SUBAPPLICATION SRV_CLIENT (* ROS 2 SRV Client *)
  (* Standard: 61499-2 *)
  (* Version 1.0, 2023-03-14, Tim Hesse *)
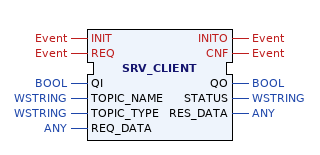
  EVENT_INPUT
    INIT; (* Initialization Request *)
    REQ; (* Normal Execution Request *)
  END_EVENT
  EVENT_OUTPUT
    INITO; (* Initialization Confirm *)
    CNF; (* Execution Confirmation *)
  END_EVENT
  VAR_INPUT
    QI : BOOL; (* Input event qualifier *)
    TOPIC_NAME : WSTRING; (* ROS 2 Topic Name *)
    TOPIC_TYPE : WSTRING; (* ROS 2 Topic Type *)
    REQ_DATA : ANY; (* Request Data *)
  END_VAR
  VAR_OUTPUT
    QO : BOOL; (* Output Event Qualifier *)
    STATUS : WSTRING; (* Service Status *)
    RES_DATA : ANY; (* Response Data *)
  END_VAR
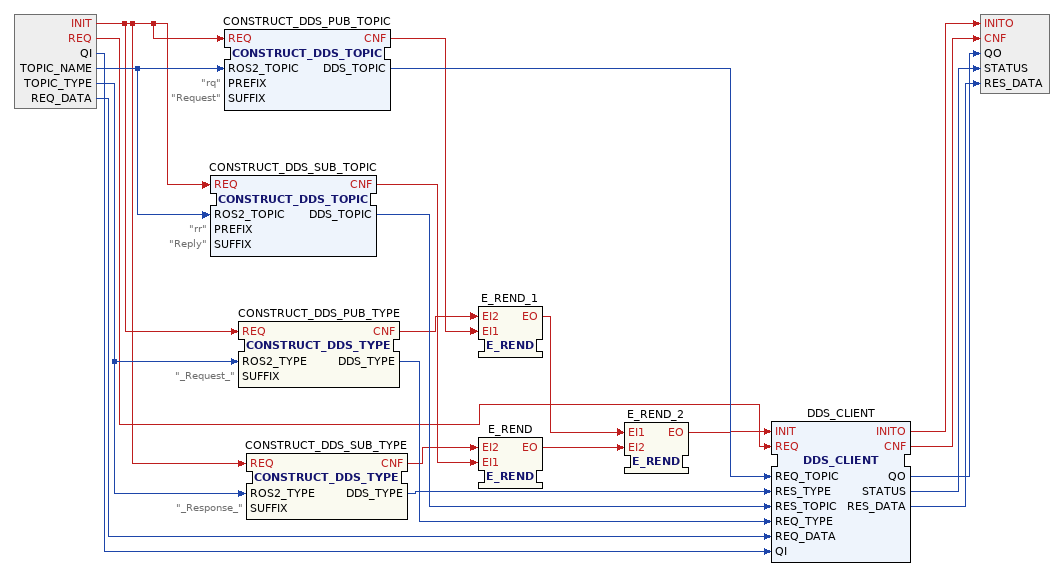
  FBS
    CONSTRUCT_DDS_PUB_TYPE : CONSTRUCT_DDS_TYPE(SUFFIX := "_Request_");
    CONSTRUCT_DDS_SUB_TYPE : CONSTRUCT_DDS_TYPE(SUFFIX := "_Response_");
    E_REND : E_REND;
    E_REND_1 : E_REND;
    E_REND_2 : E_REND;
  END_FBS
  SUBAPPS
    CONSTRUCT_DDS_PUB_TOPIC : CONSTRUCT_DDS_TOPIC(PREFIX := "rq", SUFFIX := "Request");
    CONSTRUCT_DDS_SUB_TOPIC : CONSTRUCT_DDS_TOPIC(PREFIX := "rr", SUFFIX := "Reply");
    DDS_CLIENT : DDS_CLIENT;
  END_SUBAPPS
  EVENT_CONNECTIONS
    CONSTRUCT_DDS_SUB_TYPE.CNF TO E_REND.EI2;
    CONSTRUCT_DDS_PUB_TYPE.CNF TO E_REND_1.EI2;
    INIT TO CONSTRUCT_DDS_PUB_TYPE.REQ;
    INIT TO CONSTRUCT_DDS_SUB_TYPE.REQ;
    E_REND_1.EO TO E_REND_2.EI1;
    E_REND.EO TO E_REND_2.EI2;
    INIT TO CONSTRUCT_DDS_PUB_TOPIC.REQ;
    CONSTRUCT_DDS_PUB_TOPIC.CNF TO E_REND_1.EI1;
    INIT TO CONSTRUCT_DDS_SUB_TOPIC.REQ;
    CONSTRUCT_DDS_SUB_TOPIC.CNF TO E_REND.EI1;
    DDS_CLIENT.INITO TO INITO;
    DDS_CLIENT.CNF TO CNF;
    E_REND_2.EO TO DDS_CLIENT.INIT;
    REQ TO DDS_CLIENT.REQ;
  END_CONNECTIONS
  DATA_CONNECTIONS
    TOPIC_TYPE TO CONSTRUCT_DDS_PUB_TYPE.ROS2_TYPE;
    TOPIC_TYPE TO CONSTRUCT_DDS_SUB_TYPE.ROS2_TYPE;
    TOPIC_NAME TO CONSTRUCT_DDS_PUB_TOPIC.ROS2_TOPIC;
    TOPIC_NAME TO CONSTRUCT_DDS_SUB_TOPIC.ROS2_TOPIC;
    DDS_CLIENT.QO TO QO;
    DDS_CLIENT.STATUS TO STATUS;
    DDS_CLIENT.RES_DATA TO RES_DATA;
    CONSTRUCT_DDS_PUB_TOPIC.DDS_TOPIC TO DDS_CLIENT.REQ_TOPIC;
    CONSTRUCT_DDS_SUB_TYPE.DDS_TYPE TO DDS_CLIENT.RES_TYPE;
    CONSTRUCT_DDS_SUB_TOPIC.DDS_TOPIC TO DDS_CLIENT.RES_TOPIC;
    CONSTRUCT_DDS_PUB_TYPE.DDS_TYPE TO DDS_CLIENT.REQ_TYPE;
    REQ_DATA TO DDS_CLIENT.REQ_DATA;
    QI TO DDS_CLIENT.QI;
  END_CONNECTIONS
END_SUBAPPLICATION
